RoboDK station: spiralingtest.rdk

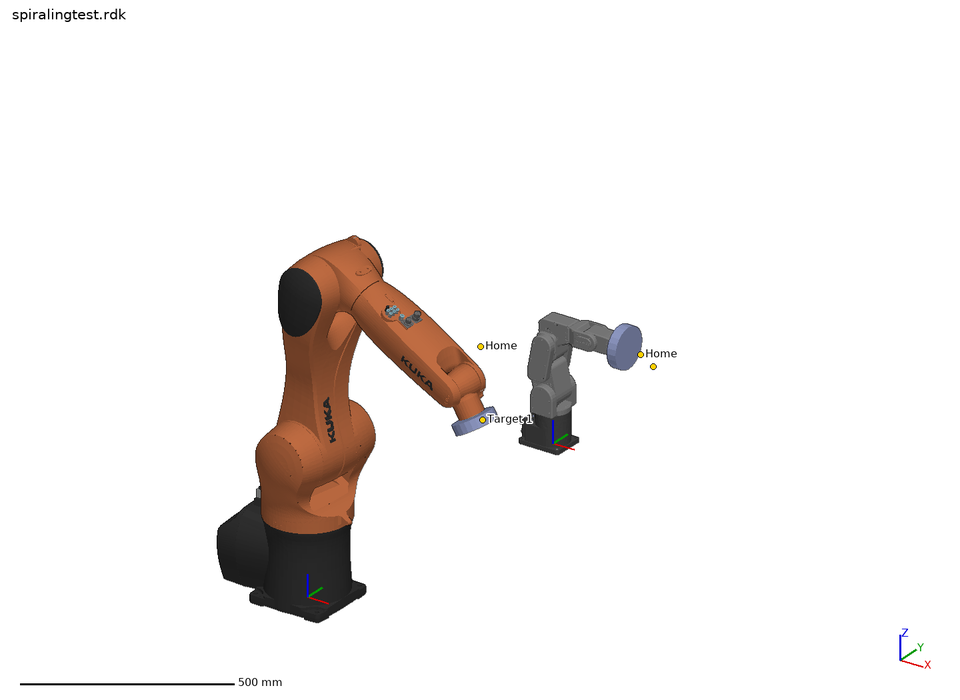
[picture v0: the station drawn from its stored meshes, robots at their saved joint values, targets as dots, program paths as lines]
Station spiralingtest (saved by RoboDK 5.5.2). Poses are relative to the parent item; angles as X-Y-Z fixed-axis rotations.
  - frame KUKA KR 6 R900 sixx Base at (0, 0, 0) mm
    - robot KUKA KR 6 R900 sixx: 6 axes, payload 6 kg, reach 901 mm, repeatability 0.03 mm, weight 52 kg
        modified DH rows (alpha deg, a mm, theta deg, d mm): 0, 0, 0, 400; -90, 25, 0, 0; 0, 455, -90, 0; -90, 35, 0, 420; 90, 0, 0, 0; -90, 0, 180, 80
        joint limits [-170, -190, -120, -185, -120, -350] to [170, 45, 156, 185, 120, 350]; home [0, -90, 90, 0, 0, 0]; saved at [6.392, -83.613, 109.185, -5.61, 34.711, 10.157]
      - tool Weld gun, TCP at (-4, 0, 371.3) mm, rotated rx 0 ry 45 rz 0 deg, size 299.9 x 60 x 318.3 mm
      - tool CrystalToolSample, TCP at (0, 0, 0) mm, size 108 x 25.4 x 108 mm, geometry from CrystalToolSample.STL
      - tool CrystalToolSample, TCP at (0, 0, 25.4) mm, size 107.9 x 25.4 x 107.9 mm, geometry from CrystalToolSample.STEP
    - target Home (Cartesian target) at (492.9, 0, 788.4) mm, rotated rx -180 ry 29.44 rz -180 deg; joints [0, -138.016, 114.252, 0, 39.328, 0] of KUKA KR 6 R900 sixx
    - target Target 1 (Cartesian target) at (500, 0, 600) mm, rotated rx -180 ry 30 rz 180 deg; joints [0, -85.787, 113.228, 0, 32.559, 0] of KUKA KR 6 R900 sixx
  - Python program DoWeld (listed below)
  - Python program Prog2 (listed below)
  - Python program Prog3 (listed below)
  - Python program Prog4 (listed below)
  - frame Mecademic Meca500 R3 Base at (0, 1000, 0) mm
    - robot Mecademic Meca500 R3: 6 axes
        modified DH rows (alpha deg, a mm, theta deg, d mm): 0, 0, 0, 135; -90, 0, -90, 0; 0, 135, 0, 0; -90, 38, 0, 120; 90, 0, 0, 0; -90, 0, 180, 70
        joint limits [-175, -70, -135, -170, -115, -720] to [175, 90, 70, 170, 115, 720]; home [0, 0, 0, 0, 0, 0]; saved at [0, 0, 0, 0, 0, 0]
      - tool CrystalToolSample, TCP at (0, 0, 25.4) mm, size 107.9 x 25.4 x 107.9 mm, geometry from CrystalToolSample.STEP
      - target Home (Cartesian target) at (8, 0, 60) mm; joints [0, -138.016, 114.252, 0, 39.328, 0] of KUKA KR 6 R900 sixx
      - target Target 1 (Cartesian target) at (58, 50, 60) mm; joints [0, -85.787, 113.228, 0, 32.559, 0] of KUKA KR 6 R900 sixx
    - Python program Prog3 (listed below)

--- Python program DoWeld ---
from robolink import *    # API to communicate with RoboDK
from robodk import *      # robodk robotics toolbox

# Any interaction with RoboDK must be done through RDK:
RDK = Robolink()

# get the robot by name:
robot = RDK.Item('', ITEM_TYPE_ROBOT)

# get the home target and the welding targets:
home = RDK.Item('Home')
target = RDK.Item('Target 1')

# get the pose of the target (4x4 matrix representing position and orientation):
poseref = target.Pose()

# move the robot to home, then to the Target 1:
robot.MoveJ(home)
robot.MoveJ(target)

# make an hexagon around the Target 1:
for i in range(7):
    ang = i*2*pi/6 #angle: 0, 60, 120, ...
    posei = poseref*rotz(ang)*transl(200,0,0)*rotz(-ang)
    robot.MoveL(posei)
    print(posei)

# move back to the center, then home:
robot.MoveL(target)
robot.MoveJ(home)

--- Python program Prog2 ---
from robodk.robolink import *       # import the robolink library (bridge with RoboDK)
RDK = Robolink()                    # establish a link with the simulator
robot = RDK.Item('KUKA KR 6 R900 sixx')      # retrieve the robot by name
#robot.setJoints([0,-115,109,0,50,0])# set all robot axes to zero

home = RDK.Item('Home')
target = RDK.Item('Target 1')# retrieve the Target item
robot.MoveJ(home)
robot.MoveJ(target)                 # move the robot to the target

# calculate a new approach position 100 mm along the Z axis of the tool with respect to the target
from robodk.robomath import *       # import the robotics toolbox
approach = target.Pose()*transl(-200,0,0)
robot.MoveL(approach)          # linear move to the approach position
approach = target.Pose()*transl(-200,100,0)
robot.MoveL(approach)

--- Python program Prog3 ---
"""
Created on Thu Jan 19 18:43:18 2023

@author: westj
"""
from robodk.robolink import *       # import the robolink library (bridge with RoboDK)
RDK = Robolink()
from robodk.robomath import *
import math
import numpy as np
import matplotlib.pyplot as plt

class Spiral:
    def __init__(self,x0:float,y0:float,points:float) -> None:
        self.x0=x0 #x offset
        self.y0=y0 #y offset
        self.points=points

    def build(self, radius:float, spacing:float):
        revs=radius/spacing            #calc number of revolutions
        k=spacing/(2*np.pi)
        theta=np.array(np.linspace(0,revs*2*np.pi,self.points)) #how many points and angle coord
        r=k * theta                       #radius coord
        x=(r*np.cos(theta)+self.x0)
        y=(r*np.sin(theta)+self.y0)             #convert to y cartesian

        return x, y #convert to x cartesian


if __name__=="__main__":
    print('Calling spiral from class')
    R=200
    S=10
    cur_spiral=Spiral(0,0,1000)
    x,y=cur_spiral.build(R,S)


 #   print(cur_spiral.build(R,S))
  #  plt.plot(x, y, color = 'red', marker = "o")
  #  plt.axis('equal')
  #  plt.show()

#______Robot Movement_________________________________________
robot = RDK.Item('KUKA KR 6 R900 sixx')
home = RDK.Item('Home')
target = RDK.Item('Target 1')# retrieve the Target item

robot.MoveJ(home)
robot.MoveJ(target)                 # move the robot to the target
#for i in x:
    #robot.MoveL(target.Pose()*transl(coord))

for i in range(len(x)):
    coord=(x[i],y[i],0)
    robot.MoveL(target.Pose()*transl(coord))
    #print(coord)
    #print('')

--- Python program Prog4 ---
__version__

--- Python program Prog3 ---
"""
Created on Thu Jan 19 18:43:18 2023

@author: westj
"""
from robodk.robolink import *       # import the robolink library (bridge with RoboDK)
RDK = Robolink()
from robodk.robomath import *
import math
import numpy as np
import matplotlib.pyplot as plt

class Spiral:
    def __init__(self,x0:float,y0:float,points:float) -> None:
        self.x0=x0 #x offset
        self.y0=y0 #y offset
        self.points=points

    def build(self, radius:float, spacing:float):
        revs=radius/spacing            #calc number of revolutions
        k=spacing/(2*np.pi)
        theta=np.array(np.linspace(0,revs*2*np.pi,self.points)) #how many points and angle coord
        r=k * theta                       #radius coord
        x=(r*np.cos(theta)+self.x0)
        y=(r*np.sin(theta)+self.y0)             #convert to y cartesian

        return x, y #convert to x cartesian


if __name__=="__main__":
    print('Calling spiral from class')
    R=200
    S=10
    cur_spiral=Spiral(0,0,1000)
    x,y=cur_spiral.build(R,S)


 #   print(cur_spiral.build(R,S))
  #  plt.plot(x, y, color = 'red', marker = "o")
  #  plt.axis('equal')
  #  plt.show()

#______Robot Movement_________________________________________
robot = RDK.Item('KUKA KR 6 R900 sixx')
home = RDK.Item('Home')
target = RDK.Item('Target 1')# retrieve the Target item

robot.MoveJ(home)
robot.MoveJ(target)                 # move the robot to the target
#for i in x:
    #robot.MoveL(target.Pose()*transl(coord))

for i in range(len(x)):
    coord=(x[i],y[i],0)
    robot.MoveL(target.Pose()*transl(coord))
    #print(coord)
    #print('')
